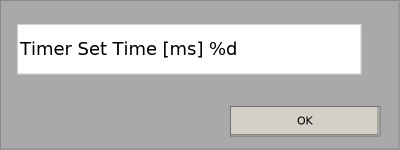
VISUALIZATION DialogTimer_HeaterOff  // 400x150
    Button (230,106 150x30), "OK"
        OnMouseClick: CloseDialog Dialog=DialogTimer_HeaterOff, Result=OK, NumpadKeypadSet=True
    Textfield (17,24 344x50), "Timer Set Time [ms] %d", text variable: PersistentStruct.TimerHotWeldingOff
        OnMouseClick: write the text variable via Edit
END_VISUALIZATION

(* stored: Version 1.1.0.1, ProductVersion 3.1.4024.3
   Visu DialogTimer_HeaterOff: Id {abb9f5c6-5d1e-46d4-93e5-20eb9eea165b} *)
